{attribute 'qualified_only'}
{attribute 'strict'}
{attribute 'to_string'}
TYPE eWifiSecurityTypes :
(
	none := 0,
	PSK2 := 1,
	SAE  := 2,
	SAE_mixed := 3,
	PSK := 4	
);
END_TYPE

(* stored: Version 1.1.0.1, ProductVersion 3.1.4026.18
   DUT eWifiSecurityTypes: Id {bd360ac4-4bae-4ead-a59e-b02922be38ca} *)
